INTERFACE I_ChunkedResponsesMiddlewareConfig

END_INTERFACE

(* stored: Version 1.1.0.1, ProductVersion 3.1.4024.12
   Itf I_ChunkedResponsesMiddlewareConfig: Id {c5d9e905-2a9d-4090-afd5-fe76d89ace34} *)
